Staubli VAL3: deb230405.dtx

jointRx jstart
mdesc mNomSpeed
